# EPICS substitutions: gigeApp/Db/pluginHDF5.substitutions
#
# pluginHDF5.substitutions
#

file NDPluginBase.template
{
	{
	P=$(CAM):,
	R=HDF5:,
	PORT=$(CAM_PORT).HDF5,
	ADDR=0,
	TIMEOUT=1,
	NDARRAY_PORT=$(PLUGIN_SRC),
	NDARRAY_ADDR=0
	}
}

file NDFile.template
{
	{
	P=$(CAM):,
	R=HDF5:,
	PORT=$(CAM_PORT).HDF5,
	ADDR=0,
	TIMEOUT=1
	}
}

file NDFileHDF5.template
{
	{
	P=$(CAM):,
	R=HDF5:,
	PORT=$(CAM).HDF5,
	ADDR=0,
	TIMEOUT=1
	}
}
